PROGRAM FB_RoomController_Test_CFC
VAR
	fbRoomController	:	FB_RoomController;
	fbLight01			:	FB_MySpecialDimmingLight;
	fbLight02			:	FB_DelayedLight;
	fbLight03			:	FB_DimmingLight;
	bAllOn				:	BOOL := FALSE;
	bAllOff				:	BOOL;
	bAllCallMinLevel	:	BOOL;
	aControlLevel		:	ARRAY [1..3] OF BOOL;
	aDimmLevel			:	ARRAY [1..3] OF BYTE;
END_VAR

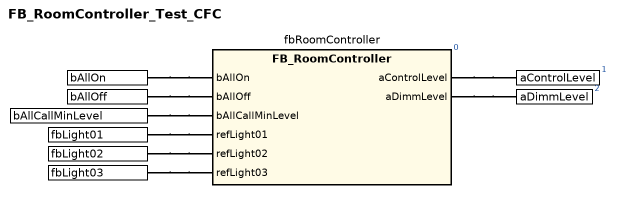
fbRoomController(
    bAllOn := bAllOn,
    bAllOff := bAllOff,
    bAllCallMinLevel := bAllCallMinLevel,
    refLight01 := fbLight01,
    refLight02 := fbLight02,
    refLight03 := fbLight03); // FB_RoomController
aControlLevel := fbRoomController.aControlLevel;
aDimmLevel := fbRoomController.aDimmLevel;

END_PROGRAM

(* stored: Version 1.1.0.1, ProductVersion 3.1.0.23
   POU FB_RoomController_Test_CFC: Id {947ac3f7-77b7-4579-afcf-2cbd7219aaa2} *)
